//{attribute 'qualified_only'}
//{attribute 'strict'}
TYPE E_Module :
(
	eModule_none := 0,
	eModule_M001,
		
	/// has to be set to last index for array bounds!
	eModule_nMaxIdx
);
END_TYPE

(* stored: Version 1.1.0.1
   DUT E_Module: Id {5b5cf293-f016-4361-a229-4d05a6bec797} *)
